// TIA Portal V20 export
FUNCTION "EM3_TeachingData" : Void   // FC79, LAD
// stored: Namespace Unit1.Em3, SetENOAutomatically false
BEGIN

REGION Network 2 (SCL): TopTape AxisX Teaching Position
   // Position 0
   "Unit1.Em3.HmiInterface".cmTopTapeAxisX.configuration.setPositions[0].position := -8.0;
   "Unit1.Em3.HmiInterface".cmTopTapeAxisX.configuration.setPositions[0].velocity := 40.0;
   "Unit1.Em3.HmiInterface".cmTopTapeAxisX.configuration.setPositions[0].acceleration := 400.0;
   "Unit1.Em3.HmiInterface".cmTopTapeAxisX.configuration.setPositions[0].deceleration := 400.0;

   // Position 1
   "Unit1.Em3.HmiInterface".cmTopTapeAxisX.configuration.setPositions[1].position := 392.72;
   "Unit1.Em3.HmiInterface".cmTopTapeAxisX.configuration.setPositions[1].velocity := 40.0;
   "Unit1.Em3.HmiInterface".cmTopTapeAxisX.configuration.setPositions[1].acceleration := 400.0;
   "Unit1.Em3.HmiInterface".cmTopTapeAxisX.configuration.setPositions[1].deceleration := 400.0;

   // Position 2
   "Unit1.Em3.HmiInterface".cmTopTapeAxisX.configuration.setPositions[2].position := 487.29;
   "Unit1.Em3.HmiInterface".cmTopTapeAxisX.configuration.setPositions[2].velocity := 40.0;
   "Unit1.Em3.HmiInterface".cmTopTapeAxisX.configuration.setPositions[2].acceleration := 400.0;
   "Unit1.Em3.HmiInterface".cmTopTapeAxisX.configuration.setPositions[2].deceleration := 400.0;

   // Position 3
   "Unit1.Em3.HmiInterface".cmTopTapeAxisX.configuration.setPositions[3].position := 200.0;
   "Unit1.Em3.HmiInterface".cmTopTapeAxisX.configuration.setPositions[3].velocity := 40.0;
   "Unit1.Em3.HmiInterface".cmTopTapeAxisX.configuration.setPositions[3].acceleration := 400.0;
   "Unit1.Em3.HmiInterface".cmTopTapeAxisX.configuration.setPositions[3].deceleration := 400.0;

   ///////////////// ZONE ////////////////////////

   // Position 9
   "Unit1.Em3.HmiInterface".cmTopTapeAxisX.configuration.setPositions[9].position := 424.0;
   "Unit1.Em3.HmiInterface".cmTopTapeAxisX.configuration.setPositions[9].velocity := 10.0;
END_REGION

REGION Network 3 (SCL): TopTape AxisY Teaching Position
   // Position 0
   "Unit1.Em3.HmiInterface".cmTopTapeAxisY.configuration.setPositions[0].position := 297.76;
   "Unit1.Em3.HmiInterface".cmTopTapeAxisY.configuration.setPositions[0].velocity := 50.0;
   "Unit1.Em3.HmiInterface".cmTopTapeAxisY.configuration.setPositions[0].acceleration := 500.0;
   "Unit1.Em3.HmiInterface".cmTopTapeAxisY.configuration.setPositions[0].deceleration := 500.0;

   // Position 1
   "Unit1.Em3.HmiInterface".cmTopTapeAxisY.configuration.setPositions[1].position := 30.8;
   "Unit1.Em3.HmiInterface".cmTopTapeAxisY.configuration.setPositions[1].velocity := 50.0;
   "Unit1.Em3.HmiInterface".cmTopTapeAxisY.configuration.setPositions[1].acceleration := 500.0;
   "Unit1.Em3.HmiInterface".cmTopTapeAxisY.configuration.setPositions[1].deceleration := 500.0;

   // Position 2
   "Unit1.Em3.HmiInterface".cmTopTapeAxisY.configuration.setPositions[2].position := 12.9;
   "Unit1.Em3.HmiInterface".cmTopTapeAxisY.configuration.setPositions[2].velocity := 50.0;
   "Unit1.Em3.HmiInterface".cmTopTapeAxisY.configuration.setPositions[2].acceleration := 500.0;
   "Unit1.Em3.HmiInterface".cmTopTapeAxisY.configuration.setPositions[2].deceleration := 500.0;


   ///////////////// ZONE ////////////////////////

   // Position 9
   "Unit1.Em3.HmiInterface".cmTopTapeAxisY.configuration.setPositions[9].position := 30.8;
   "Unit1.Em3.HmiInterface".cmTopTapeAxisY.configuration.setPositions[9].velocity := 10.0;

   // Position 10
   "Unit1.Em3.HmiInterface".cmTopTapeAxisY.configuration.setPositions[10].position := 12.9;
   "Unit1.Em3.HmiInterface".cmTopTapeAxisY.configuration.setPositions[10].velocity := 10.0;
END_REGION
END_FUNCTION
